// TIA Portal V17 export
// export: Created 2025-03-10T13:12:41.4221768Z, ExportSetting WithDefaults, DisplayName Totally Integrated Automation Portal, DisplayVersion V17 Update 8, DisplayName TIA Portal Openness, DisplayVersion V17 Update 8, DisplayName TIA Portal Version Control Interface, DisplayVersion V17, DisplayName SINAMICS Startdrive Advanced, DisplayVersion V17 SP2, DisplayName SINAMICS Startdrive G110M, G120, G120C, G120D, G120P, G115D, DisplayVersion V17 SP2, DisplayName SINAMICS Startdrive G130, G150, S120, S150, SINAMICS MV, S210, DisplayVersion V17 SP2, DisplayName STEP 7 Professional, DisplayVersion V17 Update 8, DisplayName SINUMERIK ONE STEP 7 Toolbox, DisplayVersion V17 Update 12, DisplayName SINUMERIK 840D sl STEP 7 Toolbox, DisplayVersion V17 Update 12, DisplayName STEP 7 Safety, DisplayVersion V17 Update 6, DisplayName WinCC Advanced, DisplayVersion V17 Update 8
DATA_BLOCK "DB7239_HMI_WINCC_OVERVIEW"   // DB7239
{ S7_Optimized_Access := 'TRUE' }
VERSION : 0.1
// stored: AutoNumber false, DBAccessibleFromOPCUA true, DBAccessibleFromWebserver true, IsOnlyStoredInLoadMemory false, IsRetainMemResEnabled false, IsWriteProtectedInAS false, MemoryReserve 100
   VAR
      U01_POWDER_FEEDER_1_LINE_1_OK : Bool;
      U01_POWDER_FEEDER_1_LINE_2_OK : Bool;
      U01_PF_1_LINE_1_INFINITY_FUNNEL_OK : Bool;
      U01_PF_1_LINE_1_STIRRER_OK : Bool;
      U01_PF_1_LINE_2_INFINITY_FUNNEL_OK : Bool;
      U01_PF_1_LINE_2_STIRRER_OK : Bool;
      U01_POWDER_FEEDER_OK : Bool;
      U01_PF1_L1_INF_FUNNEL_LED_STATUS : Int;   // UNIT 01 POWDER FEEDER 1 LINE 1 INFINITY FUNNEL LED STATUS
      U01_PF1_L2_INF_FUNNEL_LED_STATUS : Int;   // UNIT 01 POWDER FEEDER 1 LINE 2 INFINITY FUNNEL LED STATUS
      U02_PF1_L1_INF_FUNNEL_LED_STATUS : Int;   // UNIT 02 POWDER FEEDER 1 LINE 1 INFINITY FUNNEL LED STATUS
      U02_PF1_L2_INF_FUNNEL_LED_STATUS : Int;   // UNIT 02 POWDER FEEDER 1 LINE 2 INFINITY FUNNEL LED STATUS
      U02_PF2_L1_INF_FUNNEL_LED_STATUS : Int;   // UNIT 02 POWDER FEEDER 2 LINE 1 INFINITY FUNNEL LED STATUS
      U01_PF1_LINE_1_STATUS : Int;   // UNIT 01 POWDER FEEDER 1 LINE 1 STATUS
      U02_PF1_LINE_1_STATUS : Int;   // UNIT 02 POWDER FEEDER 1 LINE 1 STATUS
      U01_POWDER_LED_STATUS : Int;   // UNIT 01 POWDER LED STATUS
      U02_POWDER_LED_STATUS : Int;   // UNIT 02 POWDER LED STATUS
   END_VAR
BEGIN
END_DATA_BLOCK
